(* PLC project  *)

PROGRAM IdeGraphContract
  VAR
    A : INT;
    B : INT;
    C : INT;
  END_VAR

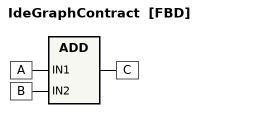
(* FBD diagram, written out as Structured Text *)
C := A + B;
END_PROGRAM
